// TIA Portal V17 export
// export: Created 2022-07-21T16:32:25.227916Z, ExportSetting WithDefaults, WithReadOnly, DisplayName Totally Integrated Automation Portal, DisplayVersion V17, DisplayName TIA Portal Openness, DisplayVersion V17, DisplayName TIA Portal Version Control Interface, DisplayVersion V17, DisplayName SINAMICS Startdrive Advanced, DisplayVersion V17, DisplayName SINAMICS Startdrive G130, G150, S120, S150, SINAMICS MV, S210, DisplayVersion V17, DisplayName SINAMICS Startdrive G110M, G120, G120C, G120D, G120P, G115D, DisplayVersion V17, DisplayName STEP 7 Professional, DisplayVersion V17, DisplayName STEP 7 Safety, DisplayVersion V17, DisplayName WinCC Advanced, DisplayVersion V17
ScreenPopup "MTR"  309x454
  ScreenLayer 
    FaceplateInstance "MTR_1" at 0,0 size 308x453  FaceplateTypeName=IO@$@MTR@$@MTR V 1.0.5
      on ClosePop: ShowPopupScreen(Name of the screen := , X coordinate := 0, Y coordinate := 0, Display mode := 0, Animation := -1, Animation speed := 1); SetTag(Tag := MTR_FacePlateNo_Visible, Value := 0)
      CM_MTR := MTR_0000
      Index := MTR_Index
      Item_number := CM_MTR_Item_numbers
      Visibility := MTR_FacePlateNo_Visible
